// TIA Portal project "EJERCICIO 7" (V11)

(* hardware
DEVICE "S7300/ET200 station_1"  SIMATIC 300-Station
   slot 0: "Perfil soporte_0"  Rail  6ES7 390-1***0-0AA0
   slot 2: "PLC_1"  CPU 313C-2 DP  6ES7 313-6CF03-0AB0  V2.6
      slot 0: "Interfaz MPI_1"  MPI
      slot 1: "Interfaz DP_1"  DP
      slot 2: "DI16/DO16_1"  DI16/DO16
      slot 4: "Contaje_1"  Counter
*)

// ===== PLC "PLC_1"  CPU 313C-2 DP =====

VAR_GLOBAL   // PLC tag table "Tabla de variables estándar"
   "MARCHA 1" AT %I0.0 : Bool;
   "MARCHA 2" AT %I0.1 : Bool;
   "LAMPARA" AT %Q0.0 : Bool;
   "Tag_1" AT %MB0 : Byte;
   "Tag_2" AT %M0.0 : Bool;
END_VAR

DATA_BLOCK "AUXILIARES"   // DB1
{ S7_Optimized_Access := 'FALSE' }
VERSION : 0.1
   VAR
      FLANCOS : Array [0..2] of Bool;
   END_VAR
BEGIN
END_DATA_BLOCK

ORGANIZATION_BLOCK "Main"   // OB1, LAD
TITLE = "Main Program Sweep (Cycle)"
{ S7_Optimized_Access := 'FALSE' }
VERSION : 0.1
   VAR_TEMP
      OB1_EV_CLASS : Byte;   // Bits 0-3 = 1 (Coming event), Bits 4-7 = 1 (Event class 1)
      OB1_SCAN_1 : Byte;   // 1 (Cold restart scan 1 of OB 1), 3 (Scan 2-n of OB 1)
      OB1_PRIORITY : Byte;   // Priority of OB Execution
      OB1_OB_NUMBR : Byte;   // 1 (Organization block 1, OB1)
      OB1_RESERVED_1 : Byte;   // Reserved for system
      OB1_RESERVED_2 : Byte;   // Reserved for system
      OB1_PREV_CYCLE : Int;   // Cycle time of previous OB1 scan (milliseconds)
      OB1_MIN_CYCLE : Int;   // Minimum cycle time of OB1 (milliseconds)
      OB1_MAX_CYCLE : Int;   // Maximum cycle time of OB1 (milliseconds)
      OB1_DATE_TIME : Date_And_Time;   // Date and time OB1 started
   END_VAR
   VAR_TEMP   // added for the SCL form of the ladder/FBD networks
      _w1 : Bool;
   END_VAR
BEGIN

REGION Network 1
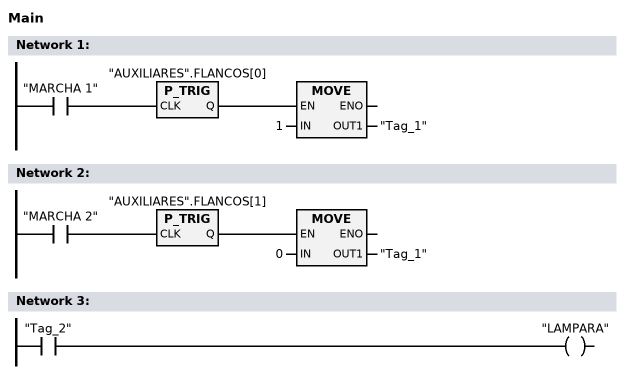
   RUNG wire#powerrail
      Contact( "MARCHA 1" )
      P_Trig( "AUXILIARES".FLANCOS[0] )
      { S7_GenerateENO := "TRUE" } Move(in := 1, out1 => "Tag_1")
   END_RUNG
   // the same network as SCL:
   #_w1 := "MARCHA 1" AND NOT "AUXILIARES".FLANCOS[0];   // rising edge
   "AUXILIARES".FLANCOS[0] := "MARCHA 1";
   IF #_w1 THEN "Tag_1" := 1; END_IF;
END_REGION

REGION Network 2
   RUNG wire#powerrail
      Contact( "MARCHA 2" )
      P_Trig( "AUXILIARES".FLANCOS[1] )
      { S7_GenerateENO := "TRUE" } Move(in := 0, out1 => "Tag_1")
   END_RUNG
   // the same network as SCL:
   #_w1 := "MARCHA 2" AND NOT "AUXILIARES".FLANCOS[1];   // rising edge
   "AUXILIARES".FLANCOS[1] := "MARCHA 2";
   IF #_w1 THEN "Tag_1" := 0; END_IF;
END_REGION

REGION Network 3
   RUNG wire#powerrail
      Contact( "Tag_2" )
      Coil( "LAMPARA" )
   END_RUNG
   // the same network as SCL:
   "LAMPARA" := "Tag_2";
END_REGION
END_ORGANIZATION_BLOCK